FUNCTION_BLOCK T_Counter IMPLEMENTS I_Counter
VAR_INPUT
END_VAR
VAR_OUTPUT
END_VAR
VAR
	count : INT;
END_VAR

METHOD IncCounter
VAR_INPUT
	Qty : INT;
END_VAR
count := count + Qty;
END_METHOD

METHOD Reset
VAR_INPUT
END_VAR
count := 0;
END_METHOD

END_FUNCTION_BLOCK

(* stored: Version 1.1.0.1, ProductVersion 3.1.4024.12
   POU T_Counter: Id {47ef5f93-3a79-4e14-9e1b-33bf32085d66}, SpecialFunc None
   Method IncCounter: Id {35cba5ef-04ae-4a72-888d-7ddff25bc476}
   Method Reset: Id {fe60da19-198a-4c4d-b542-c2433432bf80} *)
